FUNCTION_BLOCK FB_Exec_Tangential_FeedTable EXTENDS FB_ExecutorBase IMPLEMENTS I_GeometryWriter
VAR
    _NciChannel : I_NciChannel_FeedTable;
    _FeedTable  : ST_NciFeedGroupTable; 
    
    // NCI Builder z Tc2_PlcInterpolation
    fbFeedPrep  : FB_NciFeedTablePreparation;
	
	// Lokalne offsety aktualizowane co kopię nestingu
	_CurrentOffsetX : LREAL;
	_CurrentOffsetY : LREAL;
END_VAR

METHOD Abort
IF _NciChannel <> 0 THEN
    _NciChannel.Stop();
    _NciChannel.ResetChannel();
    _NciChannel.Ungroup();
END_IF
_bBusy := FALSE; _bDone := FALSE; _bError := FALSE; _uErrorID := 0; nStep := 0;
END_METHOD

METHOD AddArc : BOOL
VAR_INPUT
    TargetX    : LREAL;
    TargetY    : LREAL;
    CenterX    : LREAL;
    CenterY    : LREAL;
    Velo       : LREAL;
    Clockwise  : BOOL; 
END_VAR
VAR
    stArc : ST_NciGeoCirclePlane;
END_VAR
stArc.fEndPosX := TargetX + _CurrentOffsetX;
stArc.fEndPosY := TargetY + _CurrentOffsetY;
stArc.fCenterX := CenterX + _CurrentOffsetX;
stArc.fCenterY := CenterY + _CurrentOffsetY;
stArc.fVelo := Velo;
stArc.bClockwise := Clockwise;
stArc.nPlane := E_NciGeoPlane.E_NciGeoPlaneXY;

fbFeedPrep(
    nEntryType := E_NciEntryType.E_NciEntryTypeGeoCirclePlane,
    pEntry := ADR(stArc),
    bResetTable := FALSE,
    bResetAll := FALSE,
    stFeedGroupTable := _FeedTable
);
AddArc := NOT fbFeedPrep.bError;
END_METHOD

METHOD AddLine : BOOL
VAR_INPUT
    TargetX : LREAL;
    TargetY : LREAL;
    Velo    : LREAL;
END_VAR
VAR
    stLine : ST_NciGeoLine;
END_VAR
stLine.fEndPosX := TargetX + _CurrentOffsetX;
stLine.fEndPosY := TargetY + _CurrentOffsetY;
stLine.fVelo := Velo;

fbFeedPrep(
    nEntryType := E_NciEntryType.E_NciEntryTypeGeoLine,
    pEntry := ADR(stLine),
    bResetTable := FALSE,
    bResetAll := FALSE,
    stFeedGroupTable := _FeedTable
);
AddLine := NOT fbFeedPrep.bError;
END_METHOD

METHOD AddStartPoint : BOOL
VAR_INPUT
    TargetX : LREAL;
    TargetY : LREAL;
END_VAR
VAR
    stStart : ST_NciGeoStart;
END_VAR
stStart.fPosX := TargetX + _CurrentOffsetX;
stStart.fPosY := TargetY + _CurrentOffsetY;

fbFeedPrep(
    nEntryType := E_NciEntryType.E_NciEntryTypeGeoStart,
    pEntry := ADR(stStart),
    bResetTable := FALSE,
    bResetAll := FALSE,
    stFeedGroupTable := _FeedTable
);
AddStartPoint := NOT fbFeedPrep.bError;
END_METHOD

METHOD Clear : BOOL
VAR_INPUT
END_VAR
fbFeedPrep(
    nEntryType := E_NciEntryType.E_NciEntryTypeNone,
    pEntry := 0,
    bResetTable := TRUE,
    bResetAll := TRUE, // Czyści też modale i błędy (wg str. 315)
    stFeedGroupTable := _FeedTable
);
Clear := NOT fbFeedPrep.bError;
END_METHOD

METHOD PUBLIC CyclicLogic
VAR_INST
    localConfig   : ST_GantryXYZ_Config;
    recipeConfig  : ST_RecipeBuilder_Config;
    MaterialTopZ  : REAL;
    SafeZ         : REAL;
    TargetZ       : REAL;
END_VAR
SUPER^.CyclicLogic();

IF nStep > 0 THEN
    IF _RecipeBuilder = 0 OR _ConfigProvider = 0 OR _NciChannel = 0 THEN
        nStep := 999;
    END_IF
END_IF

CASE nStep OF
    0: 
		;
    5: 
        IF _AxisX.Enable() AND _AxisY.Enable() AND _AxisZ.Enable() AND _AxisQ.Enable() THEN
            IF _AxisX.Enabled AND _AxisY.Enabled AND _AxisZ.Enabled AND _AxisQ.Enabled 
               AND NOT _AxisX.Busy AND NOT _AxisY.Busy AND NOT _AxisQ.Busy THEN
                
                _bBusy := TRUE;
                localConfig := _ConfigProvider.Config;
                recipeConfig := _RecipeBuilder.Config;

                IF NOT recipeConfig.IsValid THEN
                    nStep := 1000;
                    RETURN;
                END_IF

                iCurrentCopyX := 1;
                iCurrentCopyY := 1;

                _AxisX.Velocity := localConfig.RapidSpeedX;
                _AxisY.Velocity := localConfig.RapidSpeedY;
                _AxisZ.Velocity := localConfig.RapidSpeedZ;
                _AxisQ.Velocity := localConfig.RapidSpeedQ;

                nStep := 8;
            END_IF
        END_IF

8: 
        localConfig := _ConfigProvider.Config;
		// Wyliczamy aktualny offset dla tej konkretnej kopii (Nesting + GlobalOffset maszyny)
		_CurrentOffsetX := (iCurrentCopyX - 1) * _RecipeBuilder.FootprintX + localConfig.GlobalOffsetX;
		_CurrentOffsetY := (iCurrentCopyY - 1) * _RecipeBuilder.FootprintY + localConfig.GlobalOffsetY;
		
		// PRZEBUDOWUJEMY TABELĘ DLA OBECNEJ KOPII
		_RecipeBuilder.Build();
		nStep := 85;

	85:
		// Czekamy na koniec budowania (Build() jest synchroniczny więc zajmie max 1 cykl)
		IF _RecipeBuilder.Done THEN
			// Odświeżamy config z buildera, bo NciStartX na pewno został przeliczony
			recipeConfig := _RecipeBuilder.Config;
			
			// NciStartX jest lokalny, MoveToXY z klasy bazowej doda Nesting + Global (czyli ustawi nas idealnie w AddStartPoint)
			MoveToXY(recipeConfig.NciStartX, recipeConfig.NciStartY, 0.0, 0.0);
			_AxisQ.MoveAbsolute(0.0, 0);
			nStep := 9;
		ELSIF _RecipeBuilder.Error THEN
			nStep := 999;
		END_IF

    9: 
        IF _AxisX.Error OR _AxisY.Error OR _AxisZ.Error OR _AxisQ.Error THEN
            nStep := 999;
        ELSIF _AxisX.InPosition AND _AxisY.InPosition AND NOT _AxisQ.Busy THEN
            localConfig := _ConfigProvider.Config;
            MaterialTopZ := localConfig.GlobalOffsetZ + localConfig.RawBoardZ;
            SafeZ := MaterialTopZ + localConfig.SafeClearanceZ;
            IF _AxisZ.MoveAbsolute(SafeZ, 0) THEN
                nStep := 10;
            END_IF
        END_IF

    10: 
        IF _AxisZ.Error THEN
            nStep := 999;
        ELSIF _AxisZ.InPosition THEN
            nStep := 20;
        END_IF

    20: 
        _NciChannel.BuildGroup();
        nStep := 30;

    30: 
        IF _NciChannel.ChannelError THEN
            nStep := 999;
        ELSIF _NciChannel.IsGrouped THEN
            TargetZ := MaterialTopZ - recipeConfig.GrooveDepthZ;
            _AxisZ.Velocity := localConfig.GroovingSpeedZ;
			IF  _AxisZ.MoveAbsolute(TargetZ, 0) THEN
				nStep := 35;
			END_IF
        END_IF

    35: 
        IF _AxisZ.Error THEN
            nStep := 999;
        ELSIF _AxisZ.InPosition THEN
            _NciChannel.StartFeedTable(stTable := THIS^._FeedTable); 
            nStep := 40;
        END_IF

    40: 
        IF _NciChannel.ChannelError THEN
            nStep := 999;
        ELSIF _NciChannel.IsFeedingDone THEN
            nStep := 50;
        END_IF

    50: 
        IF _NciChannel.ChannelError THEN
            nStep := 999;
        ELSIF _NciChannel.IsChannelDone THEN
            _AxisZ.Velocity := localConfig.RapidSpeedZ;
            _AxisZ.MoveAbsolute(SafeZ, 0);
            nStep := 55;
        END_IF

    55:
        IF _AxisZ.Error THEN
            nStep := 999;
        ELSIF _AxisZ.InPosition THEN
            _NciChannel.ResetChannel();
            nStep := 80;
        END_IF

    80: 
        _NciChannel.Ungroup();
        nStep := 90;

    90: 
        IF NOT _NciChannel.IsGrouped THEN
            nStep := 110;
        END_IF

    110:
        iCurrentCopyX := iCurrentCopyX + 1;
        IF iCurrentCopyX > _RecipeBuilder.ActualCopiesX THEN
            iCurrentCopyX := 1;
            iCurrentCopyY := iCurrentCopyY + 1;
            IF iCurrentCopyY > _RecipeBuilder.ActualCopiesY THEN
                nStep := 1000;
            ELSE
                nStep := 8;
            END_IF
        ELSE
            nStep := 8;
        END_IF

    999: 
        _bBusy := FALSE;
        _bError := TRUE;
        _bDone := FALSE;
        _uErrorID := _NciChannel.ChannelErrorId;
        _NciChannel.Ungroup();
        nStep := 0;

    1000: 
        _bBusy := FALSE;
        _bDone := TRUE;
        nStep := 0;
END_CASE
END_METHOD

METHOD EnableTangentialFollowing : BOOL
VAR
    stTf : ST_NciTangentialFollowingDesc;
END_VAR
stTf.bTangOn := TRUE;
stTf.nTangAxis := E_NciAxesInGroup.Q1Axis;
stTf.nPathAxis1 := E_NciAxesInGroup.XAxis;
stTf.nPathAxis2 := E_NciAxesInGroup.YAxis;
stTf.fOffset := -90.0;
stTf.fCriticalAngle1 := 90.0; 
stTf.nTfBehavior := E_TangentialFollowingBehavior.E_TfIngoreAll; // Uwaga na literówkę Beckhoffa!

fbFeedPrep(
    nEntryType := E_NciEntryType.E_NciEntryTypeTfDesc,
    pEntry := ADR(stTf),
    bResetTable := FALSE,
    bResetAll := FALSE,
    stFeedGroupTable := _FeedTable
);
EnableTangentialFollowing := NOT fbFeedPrep.bError;
END_METHOD

METHOD EndTable : BOOL
VAR
    stEnd : ST_NciEndOfTables;
END_VAR

fbFeedPrep(
    nEntryType := E_NciEntryType.E_NciEntryTypeEndOfTables,
    pEntry := ADR(stEnd),
    bResetTable := FALSE,
    bResetAll := FALSE,
    stFeedGroupTable := _FeedTable
);
EndTable := NOT fbFeedPrep.bError;
END_METHOD

PROPERTY NciChannel : I_NciChannel_FeedTable
GET
NciChannel := _NciChannel;
END_GET
SET
_NciChannel := NciChannel;
END_SET
END_PROPERTY

END_FUNCTION_BLOCK

(* stored: Version 1.1.0.1, ProductVersion 3.1.4024.15
   POU FB_Exec_Tangential_FeedTable: Id {e1b2c3d4-e5f6-4789-9999-000000000040}, SpecialFunc None
   Method Abort: Id {e1b2c3d4-e5f6-4789-9999-000000000042}
   Method AddArc: Id {af788716-9307-40d3-8fa3-1e39a3e2ad04}
   Method AddLine: Id {de37e77a-59fa-4e4f-b465-dfe20df19cd8}
   Method AddStartPoint: Id {55a012b2-5afc-4c4d-8025-2901f3448d7b}
   Method Clear: Id {ce1afe41-d722-4a51-b756-4addb08a67f1}
   Method CyclicLogic: Id {e1b2c3d4-e5f6-4789-9999-000000000041}
   Method EnableTangentialFollowing: Id {d2004b92-6a97-4549-b0d7-74a42dd1632f}
   Method EndTable: Id {65428bc6-7970-4afa-a4f2-edf109d35f22}
   Property NciChannel: Id {e1b2c3d4-e5f6-4789-9999-000000000043}
   Get Get: Id {e1b2c3d4-e5f6-4789-9999-000000000044}
   Set Set: Id {e1b2c3d4-e5f6-4789-9999-000000000045} *)
